// TIA Portal V15.1 export
// export: Created 2020-06-12T07:35:43.9599609Z, ExportSetting None, DisplayName Totally Integrated Automation Portal, DisplayVersion V15.1, DisplayName TIA Portal Openness, DisplayVersion V15.1, DisplayName STEP 7 Professional, DisplayVersion V15.1, DisplayName STEP 7 Safety, DisplayVersion V15.1, DisplayName WinCC Advanced, DisplayVersion V15.1
FUNCTION "PORT_ECC" : Void   // FC902, FBD
TITLE = Power Ram Clamping
{ S7_Optimized_Access := 'FALSE' }
// stored: AutoNumber false, SetENOAutomatically False
   VAR_TEMP
      tReady : Bool;
      _no_pos : Bool;
      _lock_melt : Bool;
      _cls : Bool;
      _opn : Bool;
   END_VAR
BEGIN

REGION Network 1: ECC is ready
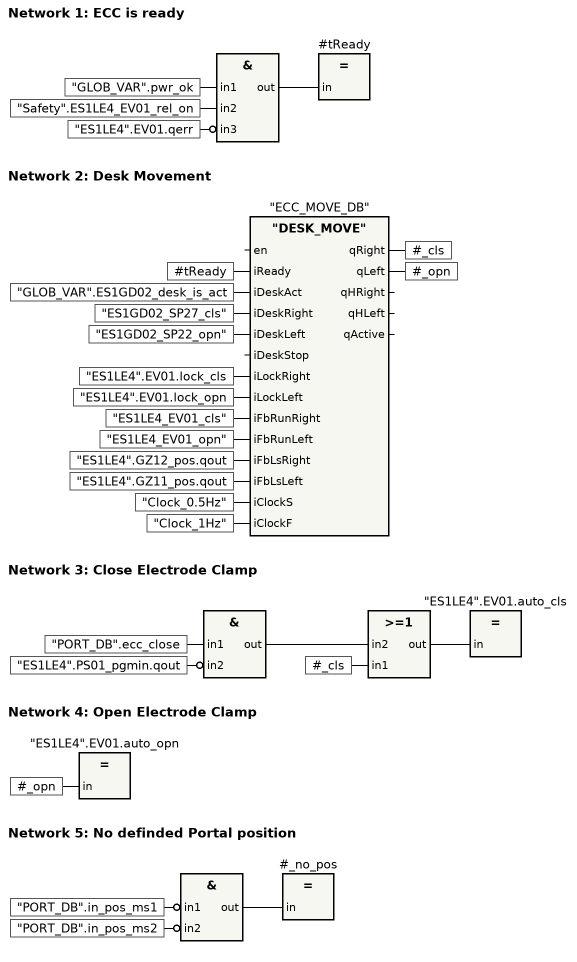
   #tReady := "GLOB_VAR".pwr_ok AND "Safety".ES1LE4_EV01_rel_on AND NOT "ES1LE4".EV01.qerr;
END_REGION

REGION Network 2: Desk Movement
   "ECC_MOVE_DB"(iReady := #tReady,   // "DESK_MOVE"
                 iDeskAct := "GLOB_VAR".ES1GD02_desk_is_act,
                 iDeskRight := "ES1GD02_SP27_cls",
                 iDeskLeft := "ES1GD02_SP22_opn",
                 iLockRight := "ES1LE4".EV01.lock_cls,
                 iLockLeft := "ES1LE4".EV01.lock_opn,
                 iFbRunRight := "ES1LE4_EV01_cls",
                 iFbRunLeft := "ES1LE4_EV01_opn",
                 iFbLsRight := "ES1LE4".GZ12_pos.qout,
                 iFbLsLeft := "ES1LE4".GZ11_pos.qout,
                 iClockS := "Clock_0.5Hz",
                 iClockF := "Clock_1Hz",
                 qRight => #_cls,
                 qLeft => #_opn);
END_REGION

REGION Network 3: Close Electrode Clamp
   "ES1LE4".EV01.auto_cls := ("PORT_DB".ecc_close AND NOT "ES1LE4".PS01_pgmin.qout) OR #_cls;
END_REGION

REGION Network 4: Open Electrode Clamp
   "ES1LE4".EV01.auto_opn := #_opn;
END_REGION

REGION Network 5: No definded Portal position
   #_no_pos := NOT "PORT_DB".in_pos_ms1 AND NOT "PORT_DB".in_pos_ms2;
END_REGION

REGION Network 6: Open Clamp Lock
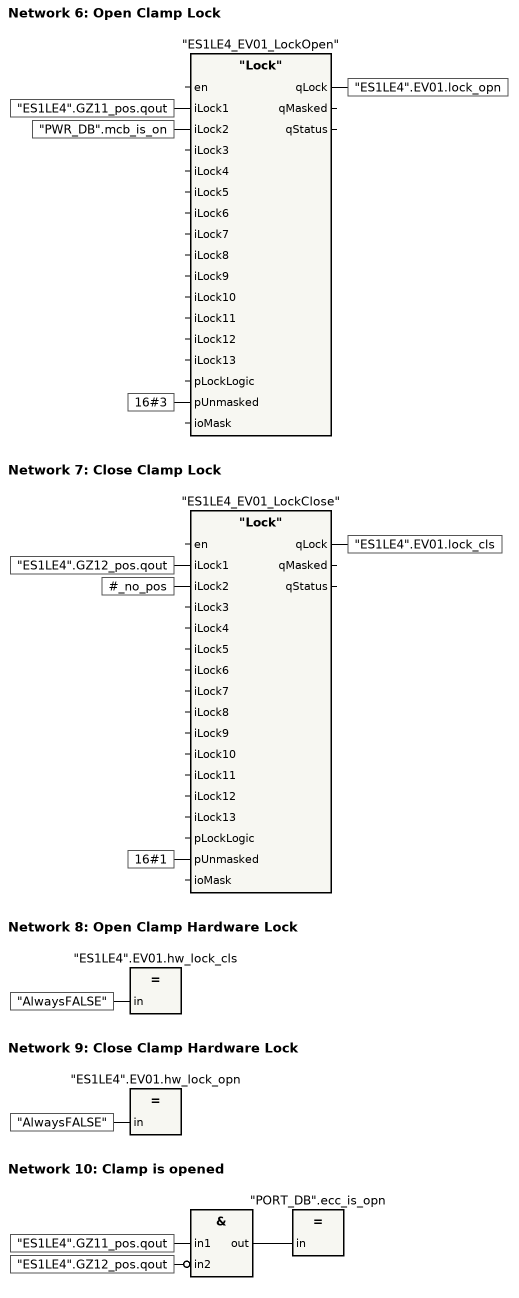
   "ES1LE4_EV01_LockOpen"(iLock1 := "ES1LE4".GZ11_pos.qout,   // "Lock"
                          iLock2 := "PWR_DB".mcb_is_on,
                          pUnmasked := 16#3,
                          qLock => "ES1LE4".EV01.lock_opn);
END_REGION

REGION Network 7: Close Clamp Lock
   "ES1LE4_EV01_LockClose"(iLock1 := "ES1LE4".GZ12_pos.qout,   // "Lock"
                           iLock2 := #_no_pos,
                           pUnmasked := 16#1,
                           qLock => "ES1LE4".EV01.lock_cls);
END_REGION

REGION Network 8: Open Clamp Hardware Lock
   "ES1LE4".EV01.hw_lock_cls := "AlwaysFALSE";
END_REGION

REGION Network 9: Close Clamp Hardware Lock
   "ES1LE4".EV01.hw_lock_opn := "AlwaysFALSE";
END_REGION

REGION Network 10: Clamp is opened
   "PORT_DB".ecc_is_opn := "ES1LE4".GZ11_pos.qout AND NOT "ES1LE4".GZ12_pos.qout;
END_REGION

REGION Network 11: Clamp closed
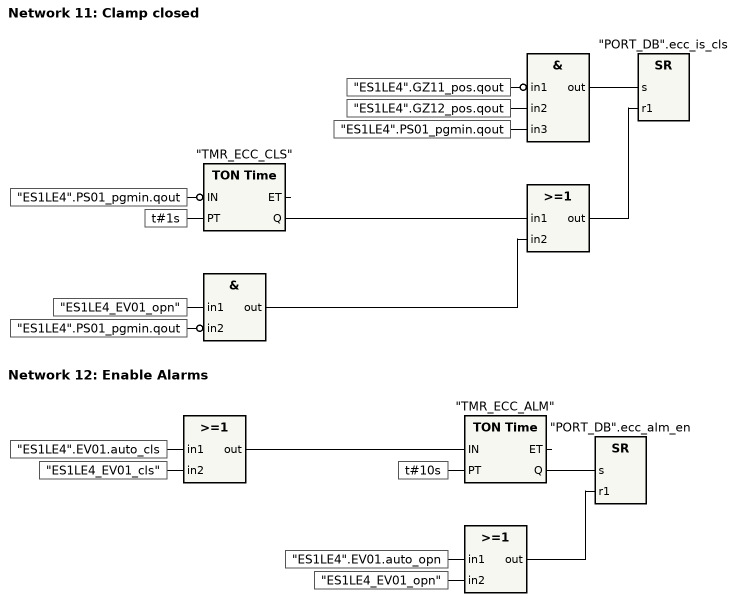
   "TMR_ECC_CLS".TON(IN := NOT "ES1LE4".PS01_pgmin.qout, PT := t#1s);
   IF NOT "ES1LE4".GZ11_pos.qout AND "ES1LE4".GZ12_pos.qout AND "ES1LE4".PS01_pgmin.qout THEN
       "PORT_DB".ecc_is_cls := TRUE;   // SR flip-flop
   END_IF;
   IF "TMR_ECC_CLS".Q OR ("ES1LE4_EV01_opn" AND NOT "ES1LE4".PS01_pgmin.qout) THEN
       "PORT_DB".ecc_is_cls := FALSE;
   END_IF;
END_REGION

REGION Network 12: Enable Alarms
   "TMR_ECC_ALM".TON(IN := "ES1LE4".EV01.auto_cls OR "ES1LE4_EV01_cls", PT := t#10s);
   IF "TMR_ECC_ALM".Q THEN
       "PORT_DB".ecc_alm_en := TRUE;   // SR flip-flop
   END_IF;
   IF "ES1LE4".EV01.auto_opn OR "ES1LE4_EV01_opn" THEN "PORT_DB".ecc_alm_en := FALSE; END_IF;
END_REGION
END_FUNCTION
